FUNCTION_BLOCK FB_SystemControl
VAR_IN_OUT
	st_params								: ST_System_params;
	st_calibration							: ST_System_calibration;
	monitor								   	: ST_System_Monitor;
	control									: ST_System_Control;
END_VAR

VAR
	//fbs
	b_calibrationRunning					: BOOL;
	PowerControl							: FB_PowerControl;
	GenGridControl							: FB_GenGridController;
	r_trigStoreMachineSettings				: R_TRIG;
	
	b_skipPowerTest								: BOOL := TRUE;
	b_StoreMachineSettings						: BOOL;
	b_loadonly									: BOOL;
	sMessage									: STRING;	

	buffer										: ARRAY [0..24] OF WORD;		

END_VAR

VAR_OUTPUT
	toSystem								: ST_System_set();
END_VAR
VAR // added by the converter: edge detectors and wires of the graphical bodies
    _rt1, _rt2, _rt3 : R_TRIG;
    _w1, _w2 : BOOL;
END_VAR

//call methods
CalculateEfficiency(
	powerstack := monitor.powerstack, 
	powermonitor := monitor.powermonitor, 
	system := monitor.system,
	battery := monitor.battery);
	
FillSystemMonitoringVars();

MapUsercontrolsToSystemVars();

GetEvents();

//store machine settings
r_trigStoreMachineSettings(CLK := settings.Save OR settings.Load);
IF r_trigStoreMachineSettings.Q THEN
	b_StoreMachineSettings := TRUE;
END_IF

IF b_StoreMachineSettings AND_THEN storeSettings(TRUE, settings.Save) THEN;
	b_StoreMachineSettings := FALSE;
END_IF

//calibration script
IF NOT st_calibration.Powerstack.Slave.b_StartCalibration THEN
	PowerstackCalibration(start := st_calibration.Powerstack.Master.b_StartCalibration, skippowertest := b_skipPowerTest, loadonly := b_loadonly,   
		powerstack := monitor.powerstack,
		powermoduleCalib := st_calibration.Powerstack.Master,
		PMeasured := monitor.powermonitor.OutputField.ar_ActivePower[0],
		QMeasured := monitor.powermonitor.OutputField.ar_ReactivePower[0],
		sMessage => sMessage);
ELSIF NOT st_calibration.Powerstack.Master.b_StartCalibration THEN
	PowerstackCalibration(start := st_calibration.Powerstack.Slave.b_StartCalibration, skippowertest := b_skipPowerTest, loadonly := b_loadonly,   
		powerstack := monitor.powerstack,
		powermoduleCalib := st_calibration.Powerstack.Slave,
		PMeasured := monitor.powermonitor.OutputField.ar_ActivePower[0],
		QMeasured := monitor.powermonitor.OutputField.ar_ReactivePower[0],
		sMessage => sMessage);
END_IF
b_calibrationRunning := settings.Calibration.Powerstack.Master.b_StartCalibration OR settings.Calibration.Powerstack.Slave.b_StartCalibration;


UpdateSystemTime();

METHOD PRIVATE CalculateEfficiency : BOOL
VAR_IN_OUT
	powerstack 				: st_Powerstack_get;
	powermonitor			: st_powermonitor_get;
	system					: ST_system_get;
	battery					: ST_bms_get;
END_VAR

VAR_INST
	r_RawEfficiency	: REAL;
	r_AverageEfficiency: REAL;
	r_RoundtripEfficiency: REAL;
	
	
	ton_SumTimer			: TON :=(PT := T#100ms);
	r_EfficiencySum			: REAL;
	w_AverageSumCounter			: WORD;
END_VAR
r_RawEfficiency := ABS(powerstack.r_DCPower) / MAX(1,ABS(powermonitor.InputField.ar_ActivePower[0] + powermonitor.OutputField.ar_ActivePower[0])) * 100;

system.r_CurrentEfficiency := LIMIT(0, r_rawEfficiency, 99.8);

//manual averaging of the last hour of operation
ton_SumTimer(IN := NOT ton_SumTimer.Q);
IF powerstack.b_StartedState AND ton_SumTimer.Q THEN
	//reset counter and sum after 3000 samples +- 5min.
	IF w_AverageSumCounter = 3000 THEN
		//increment array index to add new efficiency value until upperbound has been reached.
		r_efficiencySum := r_efficiencySum - r_AverageEfficiency + system.r_CurrentEfficiency;
	ELSE
		//add new value to the summation
		w_AverageSumCounter := w_AverageSumCounter +1;
		r_EfficiencySum := r_efficiencySum + system.r_CurrentEfficiency;
	END_IF
	
	//System average efficiency during operation
	r_AverageEfficiency := r_EfficiencySum / MAX(1, w_AverageSumCounter);
	system.r_AvgEfficiency := r_AverageEfficiency;
	r_RoundtripEfficiency := LIMIT(0, powermonitor.Inverter.r_EnergySupplied / MAX(1,powermonitor.Inverter.r_EnergyConsumed - Battery.BatteryInfo.r_RemainingDischargeEnergyNett) * 100, 99);
	System.r_RoundtripEfficiency := r_RoundtripEfficiency;
END_IF
END_METHOD

METHOD ConfigureOutputContact : BOOL
VAR_INPUT
	SignalSelect			: eOutputContactSignal;
	GensetStartStop			: BOOL;
END_VAR
CASE SignalSelect OF
	eOutputContactSignal.FireAlarm 		: ConfigureOutputContact:= monitor.protections.FireDetection.b_FireAlarm;
	eOutputContactSignal.GenStartStop 	: ConfigureOutputContact:= GensetStartStop;
END_CASE
END_METHOD

METHOD EMstop : BOOL
VAR_INPUT
END_VAR

VAR_INST
	ton_FBdelay : TON := (PT:= T#20MS);
END_VAR
EMstop := FALSE;
ton_FBdelay(IN:= TRUE);

IF ton_FBdelay.Q THEN
	ton_FBdelay.IN := FALSE;
	EMstop := TRUE;
END_IF
END_METHOD

METHOD FillSystemMonitoringVars : BOOL

VAR_INST
	st_Params_MA			: ST_CTRL_MOVING_AVERAGE_PARAMS;
	ui_filterSize			: UINT := 50;
	fb_AverageEff			: FB_CTRL_MOVING_AVERAGE;
END_VAR
monitor.b_modeSwitchEnable := monitor.system.e_State = eSystemstate.Off OR 
	monitor.system.e_State = eSystemstate.StandBy OR
	monitor.system.e_State = eSystemstate.Init OR
	monitor.system.e_State = eSystemstate.Conditioning OR
	monitor.system.e_State = eSystemstate.Transport OR 
	monitor.system.e_State = eSystemstate.Dehumidifying OR
	monitor.system.e_State = eSystemState.EMstop; 

//Effiencies
monitor.system.b_StartAllowed := 
	control.HardSettings.system.e_EarthingSystem <> 0 AND
	monitor.powerstack.b_StartEnabled AND monitor.Cooling.ui_DehumRemainingTime = 0;
monitor.system.s_SystemName := Monitor.Router.Mobile.s_EmergencySMSDevName;

CASE toSystem.powerstack.e_Powermode OF
	ePowermodes.Droop: monitor.system.e_UgridPowermode := eUgridPowermode.Droop;
	ePowermodes.DroopZeroStart: monitor.system.e_UgridPowermode := eUgridPowermode.DroopZeroStart;
	ePowermodes.Isochronous: monitor.system.e_UgridPowermode := eUgridPowermode.Isochronous;
END_CASE

CASE toSystem.powerstack.e_InverterMode OF
	eInvertermodes.Afe : 
		monitor.system.e_gridmode := eGridmode.following;
		monitor.system.e_UgridPowermode := eUgridPowermode.None;
	eInvertermodes.Microgrid : monitor.system.e_gridmode := eGridmode.forming;
END_CASE
END_METHOD

METHOD GetDiagnostics
VAR_IN_OUT
	AddError		: ARRAY [*] OF FB_AddErrorST;
	a_ActiveEvents	: ARRAY [*] OF ST_ErrorStruct;
	w_Index			: WORD;
END_VAR
GenGridControl.GetDiagnostics(AddError, a_ActiveEvents, w_Index);
PowerControl.GetDiagnostics(AddError, a_ActiveEvents, w_Index);

(*Machine name update pending*) 	AddError[w_Index](
		b_ErrorTrig				:= monitor.system.events.b_RestartRequiredMachineName,
		out_ST_Error			:= a_ActiveEvents[w_Index],
		w_ErrorID				:= 1,
		e_ObjectID				:= eObject_ID.system,
		s_Message				:= 'Machinename update pending in VDL Powernet: System restart required',
		e_sev					:= eseverity.Info
		);
	w_Index := w_Index +1;
	
(*Machine name update pending*) AddError[w_Index](
		b_ErrorTrig				:= monitor.HartingIO.b_ExtSystemShutdownRequest,
		out_ST_Error			:= a_ActiveEvents[w_Index],
		w_ErrorID				:= 2,
		e_ObjectID				:= eObject_ID.system,
		s_Message				:= 'External IO initiated system shutdown',
		e_sev					:= eseverity.NormalShutdown,
		b_autoclear				:= FALSE
		);
	w_Index := w_Index +1;
	
(*time update failed*)	AddError[w_Index](
			b_ErrorTrig				:= monitor.system.events.b_TimeUpdateFailed,
			b_SMSEnableVDL			:= FALSE,
			out_ST_Error			:= a_ActiveEvents[w_Index],
			w_ErrorID				:= 3,					
			s_Message				:= 'System time update failed',
			e_sev					:= eSeverity.info,
			b_AutoClear				:= TRUE,
			e_ErrAckAccess			:= eErrAckAccess.General
			);
		w_Index := w_Index +1;
END_METHOD

METHOD GetEvents : BOOL
VAR_INPUT
END_VAR

VAR_INST
	s_machineNameOld : STRING;
	initdone		: BOOL;
END_VAR
IF NOT initdone AND monitor.system.s_SystemName <> '' THEN
	s_machineNameOld := monitor.system.s_SystemName;
	initdone := TRUE;
END_IF

monitor.system.events.b_RestartRequiredMachineName := s_machineNameOld <> monitor.system.s_SystemName;
END_METHOD

METHOD JsonFileToStruct : BOOL
VAR_INPUT
	bExecute			: BOOL;
	sJsonPathname		: STRING := 'C:\PLC_Utility\CalData_Powerstack.json';
	sStructName			: STRING;
	pStruct				: PVOID;
	nStruct				: UDINT;
	WriteMode			: BOOL;
	
END_VAR

VAR_OUTPUT
	Busy			: BOOL;
	Error			: BOOL;
	sMessage		: STRING;
END_VAR

VAR_INST
	bEnableCreateFile 	: BOOL := TRUE;
	SfcstepPrev		: BYTE;
	SFCTransAllowed	: BOOL;
	tofSFCstepDelay	: TOF := (PT := T#20MS);
	fbFileRead 		: FB_FileRead;
	fbFileWrite		: FB_FileWrite;
	fbFileOpen		: FB_FileOpen;
	fbFileClose		: FB_FileClose;
	sErrorMessage	: STRING;
	bLoading 		: BOOL;
	ton_executedelay	: TON := (PT := T#10MS);
	SFCstep			: BYTE;
	bLoad			: BOOL;
	bError			: BOOL;
	bfileOpened		: BOOL;
	hrErrorCode		: HRESULT;
	fbJson         : FB_JsonSaxWriter;
  	fbJsonDataType : FB_JsonReadWriteDataType;
  	sJsonDoc     	: STRING(10000);
	nBytesRead		: UDINT;
	b_CreateNewFile 	: BOOL;
	bOpenExecute		: BOOL;
	bReadExecute		: BOOL;
	bWriteExecute		: BOOL;
	bCloseExecute		: BOOL;
	nModeSel			: DWORD;	
	udLength			: UDINT;
	tDelayWriting		: TON := (PT := T#50MS);
	bEnable : BOOL := FALSE;
	
END_VAR
 

IF NOT ton_executedelay.Q THEN
	sfcstep := 0;
END_IF

IF pStruct = 0 THEN
	sfcstep := 99;
	sErrorMessage := 'Invalid pointer to struct';
ELSIF nStruct = 0 THEN
	sfcstep := 99;
	sErrorMessage := 'Invalid size of struct';
END_IF

//transition delay logic.
tofSFCstepDelay(IN := SFCstep <> SFCstepPrev);
SFCTransAllowed := NOT tofSFCstepDelay.Q AND bLoading;

CASE SFCstep OF
0: //idle
bEnable := FALSE;
	bLoading := FALSE;
	bError := FALSE;
	SFCTransAllowed := FALSE;
	bOpenExecute 			:= FALSE;
	bReadExecute 			:= FALSE;
	bWriteExecute 			:= FALSE;
	bCloseExecute 			:= FALSE;
	bEnableCreateFile 		:= FALSE;
	
	ton_executedelay(IN := bExecute);
	
	IF ton_executedelay.Q THEN
		sfcstep := SEL(writemode OR b_CreateNewFile, 1, 2);
		nModeSel 		:= SEL(sfcstep = 1, FOPEN_MODEWRITE,FOPEN_MODEREAD);
		sErrorMessage := '';
		bLoading := TRUE;	
	END_IF
	
1: 	//open file
	sJsonDoc := '';
	nModeSel 				:= FOPEN_MODEREAD;
	bReadExecute 			:= FALSE;
	bWriteExecute 			:= FALSE;
	bCloseExecute 			:= FALSE;
	bOpenExecute 			:= SFCTransAllowed;
	
	
	IF bEnable THEN 
	//IF SFCTransAllowed THEN
		IF fbFileOpen.hfile <> 0 AND NOT fbFileOpen.bBusy AND NOT fbFileOpen.bError THEN
			SFCstep := 10;
			bEnable := FALSE;
		ELSIF fbFileOpen.bError THEN
			sErrorMessage := CONCAT('Error opening file: sfc step ', TO_STRING(sfcstep));
			sfcstep := SEL(bEnableCreateFile, 97, 2);
		END_IF
	END_IF
	
2: //create file if non existing
	sJsonDoc := '';
	b_createNewFile := FALSE;
	nModeSel 				:= FOPEN_MODEWRITE;
	bReadExecute 			:= FALSE;
	bWriteExecute 			:= FALSE;
	bCloseExecute 			:= FALSE;
	bOpenExecute 			:= SFCTransAllowed;

	
	IF bEnable THEN 
		IF fbFileOpen.hfile <> 0 AND NOT fbFileOpen.bBusy AND NOT fbFileOpen.bError THEN
			sErrorMessage := 'New file created';
			sJsonDoc 		:= '';
			MEMSET(ADR(sJsonDoc), 0, SIZEOF(sJsonDoc));
			SFCstep := 3;
			bEnable := FALSE;
		ELSIF fbFileOpen.bError THEN
			sErrorMessage := CONCAT('Error opening and creating file: sfc step ', TO_STRING(sfcstep));
			sfcstep := 97;
		END_IF
	END_IF
	
3: //Write current struct values to new Json string
//	IF LEN(sJsonDoc) = 0 THEN
		fbJson.ResetDocument();
		fbJsonDataType.AddJsonValueFromSymbol(fbJson, sStructName, nStruct, pStruct, hrErrorCode => hrErrorCode);
		udLength := fbJson.GetDocumentLength();
		fbJson.CopyDocument(sJsonDoc, udLength);
//	END_IF
	
	IF SFCTransAllowed THEN
		IF hrErrorCode = 0 THEN
			bError := FALSE;
			sfcstep := 4; //final step
		ELSE
			bError := TRUE;
			sErrorMessage := CONCAT('Error generating json string: SFC step ', TO_STRING(sfcstep));
			sfcstep := 97; //error step
		END_IF
	END_IF
	
4: //write json string to file
	bReadExecute 	:= FALSE;
	bOpenExecute 	:= FALSE;
	bCloseExecute 	:= FALSE;
	bWriteExecute 	:= SFCTransAllowed;
	
	IF SFCTransAllowed THEN
		IF NOT fbFileWrite.bBusy AND NOT fbFileWrite.bError THEN
			SFCstep := 97;
			bEnable := FALSE;
		ELSIF fbFileWrite.bError THEN
			sErrorMessage := CONCAT('Error writing file: sfc step ', TO_STRING(sfcstep));
			sfcstep := 97;
		END_IF
	END_IF
		
10: //Read File
	sJsonDoc 		:= '';
	bOpenExecute 	:= FALSE;
	bWriteExecute 	:= FALSE;
	bCloseExecute 	:= FALSE;
	bReadExecute 	:= SFCTransAllowed;
	
	IF SFCTransAllowed THEN
		IF NOT fbFileRead.bBusy AND NOT fbFileRead.bError THEN
			SFCstep := 11;
			bEnable := FALSE;
		ELSIF fbFileRead.bError THEN
			sErrorMessage := CONCAT('Error reading file: sfc step ', TO_STRING(sfcstep));
			sfcstep :=  97;
			b_createNewFile := bEnableCreateFile;
		END_IF
	END_IF

	
11: //Convert buffer to struct
	fbJsonDataType.SetSymbolFromJson(sJsonDoc, sStructName, nStruct, pStruct, hrErrorCode => hrErrorCode);
	
	IF SFCTransAllowed THEN
		
		IF hrErrorCode = 0 THEN
			bError := FALSE;
			sfcstep := 97; //final step
		ELSE
			bError := TRUE;
			sErrorMessage := CONCAT('Error writing file to struct: sfc step ', TO_STRING(sfcstep));
			sfcstep := 97;
			b_createNewFile := bEnableCreateFile;	
		END_IF
	END_IF

97: // file opened
	
	bWriteExecute 	:= FALSE;
	bOpenExecute 	:= FALSE;
	bReadExecute 	:= FALSE;
	bCloseExecute 	:= bfileOpened := fbFileOpen.hFile <> 0;

	
	IF SFCTransAllowed THEN
		IF NOT fbFileClose.bBusy AND NOT fbFileClose.bError THEN
			bfileOpened := FALSE;
			sfcstep := 98;
			bEnable := FALSE;
		ELSIF fbFileClose.bError THEN
			sErrorMessage := CONCAT('Error closing file ', TO_STRING(sfcstep));
			bError := TRUE;
			sfcstep := 98;
		END_IF
	END_IF
	
98: 	//feedback and reset method for next request
	IF NOT bError THEN
		sErrorMessage := 'SUCCES';
	ELSE
		Error := TRUE;
	END_IF
	bEnable := FALSE;
	bOpenExecute 		:= FALSE;
	bReadExecute 		:= FALSE;
	bWriteExecute 		:= FALSE;
	bCloseExecute 		:= FALSE;
	ton_executedelay.IN := FALSE;
	sfcstep := 99;
	
	
99: //once here, reset SFC
	IF NOT b_CreateNewFile THEN
		JsonFileToStruct := TRUE;
	END_IF
	sfcstep := 0;
END_CASE
	


fbFileOpen(sPathName:= sJsonPathname , nMode := nModeSel ,bExecute:= bOpenExecute);
fbFileWrite(hFile := fbFileOpen.hFile , pWriteBuff := ADR(sJsonDoc),bExecute := bWriteExecute , cbWriteLen := udLength);
fbFileRead(hFile := fbFileOpen.hFile, pReadBuff := ADR(sJsonDoc), cbReadLen := SIZEOF(sJsonDoc),bExecute := bReadExecute, cbRead => nBytesRead);
fbFileClose(hFile := fbFileOpen.hFile, bExecute := bCloseExecute);

IF fbFileOpen.bBusy AND bOpenExecute THEN
	bOpenExecute := FALSE;
	bEnable := TRUE;
END_IF
//	rTrigExecute(CLK := FALSE);
//	IF NOT rTrigExecute.CLK THEN
//		JsonFileToStruct := TRUE;
SFCstepPrev := SFCstep;

//output data
busy := bLoading;
sMessage := sErrorMessage;
END_METHOD

ACTION Map_ACDCchargerControls:
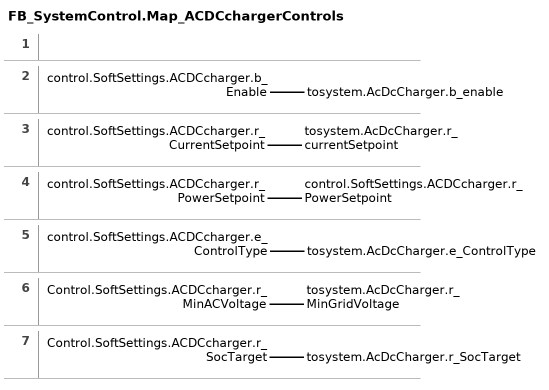
// NETWORK 1

// NETWORK 2
tosystem.AcDcCharger.b_enable := control.SoftSettings.ACDCcharger.b_Enable;

// NETWORK 3
tosystem.AcDcCharger.r_currentSetpoint := control.SoftSettings.ACDCcharger.r_CurrentSetpoint;

// NETWORK 4
control.SoftSettings.ACDCcharger.r_PowerSetpoint := control.SoftSettings.ACDCcharger.r_PowerSetpoint;

// NETWORK 5
tosystem.AcDcCharger.e_ControlType := control.SoftSettings.ACDCcharger.e_ControlType;

// NETWORK 6
tosystem.AcDcCharger.r_MinGridVoltage := Control.SoftSettings.ACDCcharger.r_MinACVoltage;

// NETWORK 7
tosystem.AcDcCharger.r_SocTarget := Control.SoftSettings.ACDCcharger.r_SocTarget;
END_ACTION

ACTION MaP_BMSControl:
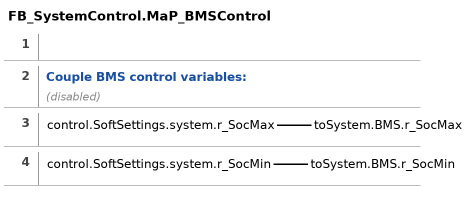
// NETWORK 1

// NETWORK 2 (disabled)
// label: Couple BMS control variables

// NETWORK 3
toSystem.BMS.r_SocMax := control.SoftSettings.system.r_SocMax;

// NETWORK 4
toSystem.BMS.r_SocMin := control.SoftSettings.system.r_SocMin;
END_ACTION

ACTION Map_DCLink:
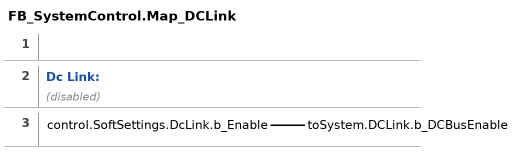
// NETWORK 1

// NETWORK 2 (disabled)
// label: Dc Link

// NETWORK 3
toSystem.DCLink.b_DCBusEnable := control.SoftSettings.DcLink.b_Enable;
END_ACTION

ACTION Map_GenCommControls:
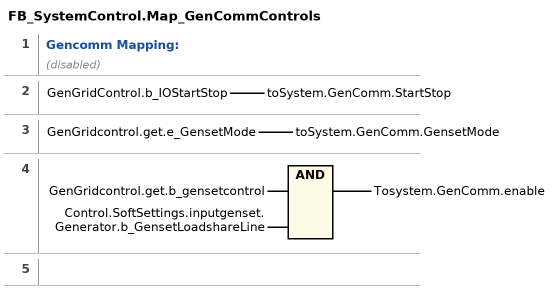
// NETWORK 1 (disabled)
// label: Gencomm Mapping

// NETWORK 2
toSystem.GenComm.StartStop := GenGridControl.b_IOStartStop;

// NETWORK 3
toSystem.GenComm.GensetMode := GenGridcontrol.get.e_GensetMode;

// NETWORK 4
Tosystem.GenComm.enable := GenGridcontrol.get.b_gensetcontrol AND Control.SoftSettings.inputgenset.Generator.b_GensetLoadshareLine;

// NETWORK 5
END_ACTION

ACTION Map_GeneralControls:
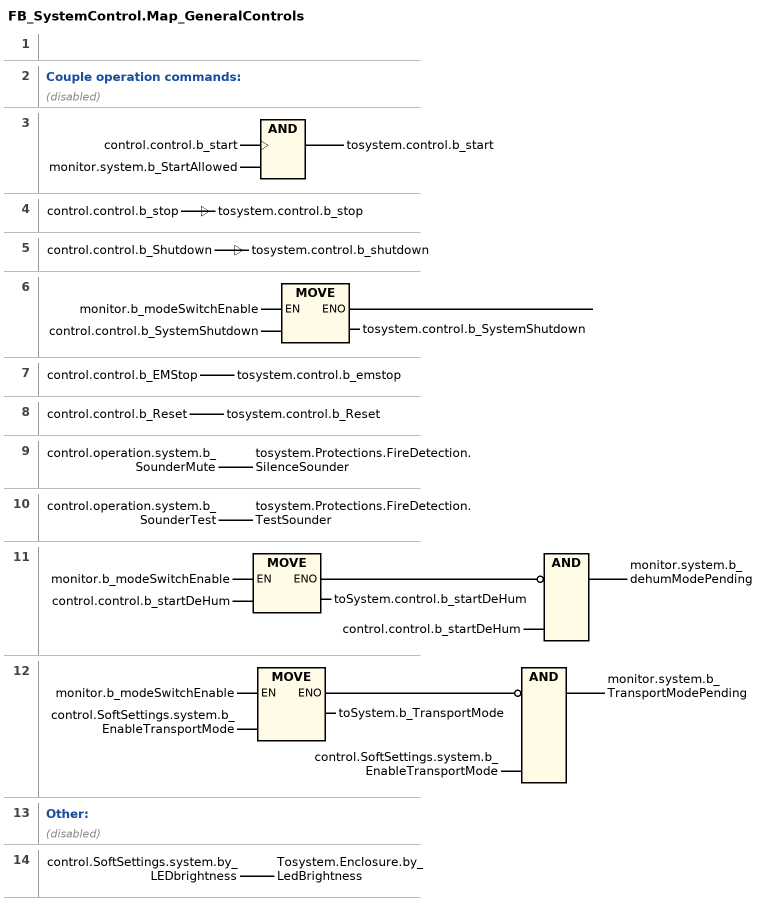
// NETWORK 1

// NETWORK 2 (disabled)
// label: Couple operation commands

// NETWORK 3
_rt1(CLK := control.control.b_start);
tosystem.control.b_start := _rt1.Q AND monitor.system.b_StartAllowed;

// NETWORK 4
_rt2(CLK := control.control.b_stop);
tosystem.control.b_stop := _rt2.Q;

// NETWORK 5
_rt3(CLK := control.control.b_Shutdown);
tosystem.control.b_shutdown := _rt3.Q;

// NETWORK 6
IF monitor.b_modeSwitchEnable THEN tosystem.control.b_SystemShutdown := control.control.b_SystemShutdown; END_IF

// NETWORK 7
tosystem.control.b_emstop := control.control.b_EMStop;

// NETWORK 8
tosystem.control.b_Reset := control.control.b_Reset;

// NETWORK 9
tosystem.Protections.FireDetection.SilenceSounder := control.operation.system.b_SounderMute;

// NETWORK 10
tosystem.Protections.FireDetection.TestSounder := control.operation.system.b_SounderTest;

// NETWORK 11
_w1 := monitor.b_modeSwitchEnable;
IF _w1 THEN toSystem.control.b_startDeHum := control.control.b_startDeHum; END_IF
monitor.system.b_dehumModePending := NOT _w1 AND control.control.b_startDeHum;

// NETWORK 12
_w2 := monitor.b_modeSwitchEnable;
IF _w2 THEN toSystem.b_TransportMode := control.SoftSettings.system.b_EnableTransportMode; END_IF
monitor.system.b_TransportModePending := NOT _w2 AND control.SoftSettings.system.b_EnableTransportMode;

// NETWORK 13 (disabled)
// label: Other

// NETWORK 14
Tosystem.Enclosure.by_LedBrightness := control.SoftSettings.system.by_LEDbrightness;
END_ACTION

ACTION Map_HartingIO:
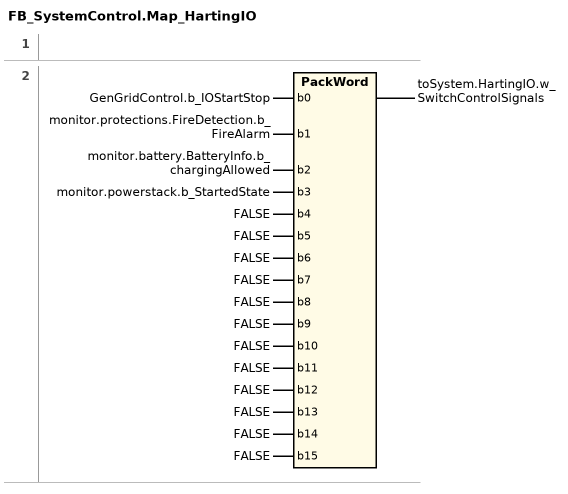
// NETWORK 1

// NETWORK 2
toSystem.HartingIO.w_SwitchControlSignals := PackWord(b0 := GenGridControl.b_IOStartStop, b1 := monitor.protections.FireDetection.b_FireAlarm, b2 := monitor.battery.BatteryInfo.b_chargingAllowed, b3 := monitor.powerstack.b_StartedState, b4 := FALSE, b5 := FALSE, b6 := FALSE, b7 := FALSE, b8 := FALSE, b9 := FALSE, b10 := FALSE, b11 := FALSE, b12 := FALSE, b13 := FALSE, b14 := FALSE, b15 := FALSE);
END_ACTION

ACTION Map_PowerstackControls:
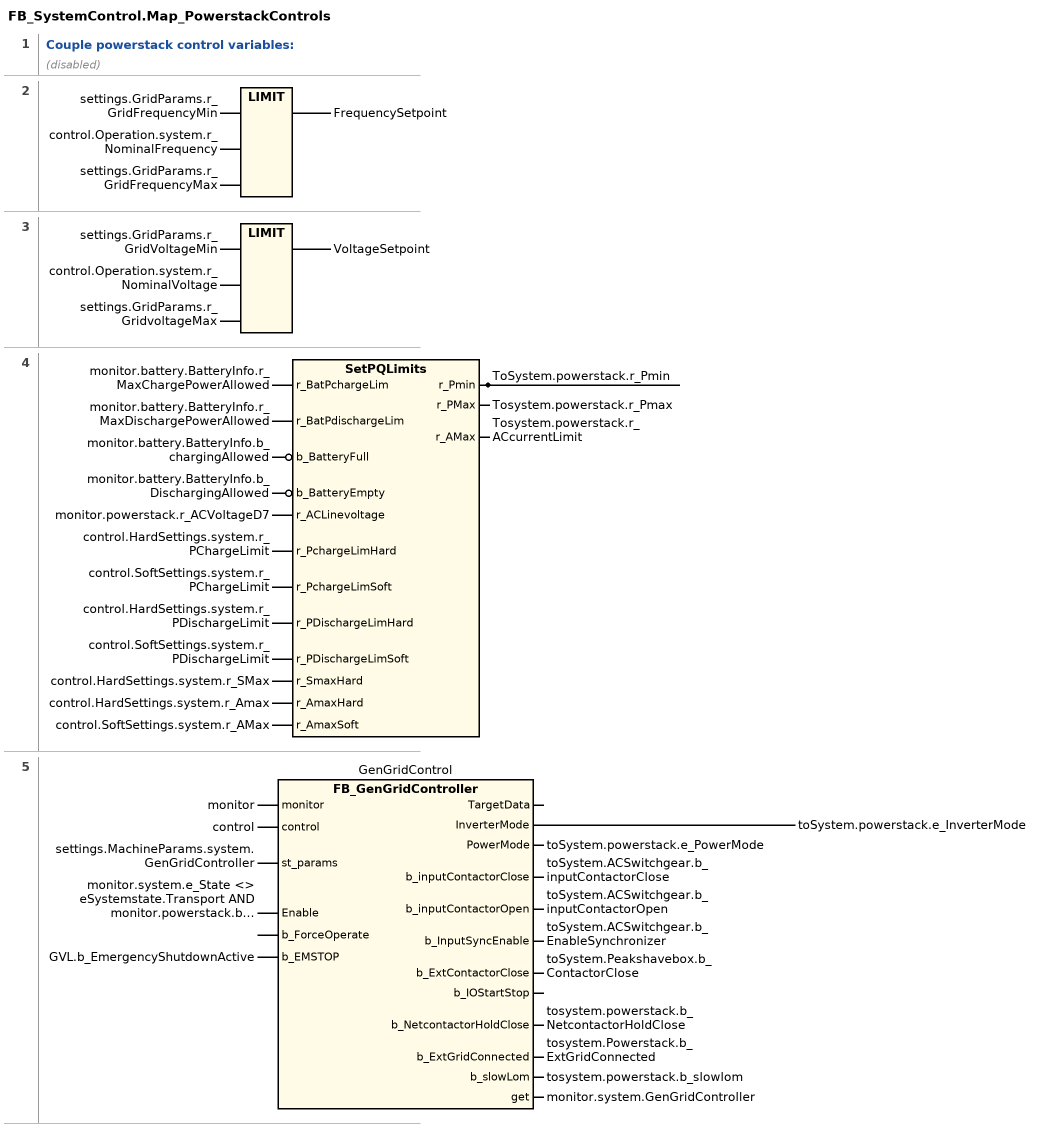
// NETWORK 1 (disabled)
// label: Couple powerstack control variables

// NETWORK 2
FrequencySetpoint := LIMIT(settings.GridParams.r_GridFrequencyMin, control.Operation.system.r_NominalFrequency, settings.GridParams.r_GridFrequencyMax);

// NETWORK 3
VoltageSetpoint := LIMIT(settings.GridParams.r_GridVoltageMin, control.Operation.system.r_NominalVoltage, settings.GridParams.r_GridvoltageMax);

// NETWORK 4
SetPQLimits(r_BatPchargeLim := monitor.battery.BatteryInfo.r_MaxChargePowerAllowed, r_BatPdischargeLim := monitor.battery.BatteryInfo.r_MaxDischargePowerAllowed, b_BatteryFull := NOT monitor.battery.BatteryInfo.b_chargingAllowed, b_BatteryEmpty := NOT monitor.battery.BatteryInfo.b_DischargingAllowed, r_ACLinevoltage := monitor.powerstack.r_ACVoltageD7, r_PchargeLimHard := control.HardSettings.system.r_PChargeLimit, r_PchargeLimSoft := control.SoftSettings.system.r_PChargeLimit, r_PDischargeLimHard := control.HardSettings.system.r_PDischargeLimit, r_PDischargeLimSoft := control.SoftSettings.system.r_PDischargeLimit, r_SmaxHard := control.HardSettings.system.r_SMax, r_AmaxHard := control.HardSettings.system.r_Amax, r_AmaxSoft := control.SoftSettings.system.r_AMax, r_Pmin => ToSystem.powerstack.r_Pmin, r_PMax => Tosystem.powerstack.r_Pmax, r_AMax => Tosystem.powerstack.r_ACcurrentLimit);

// NETWORK 5
GenGridControl(
    monitor := monitor,
    control := control,
    st_params := settings.MachineParams.system.GenGridController,
    Enable := monitor.system.e_State <> eSystemstate.Transport AND monitor.powerstack.b_ControlEnabled,
    b_EMSTOP := GVL.b_EmergencyShutdownActive,
    PowerMode => toSystem.powerstack.e_PowerMode,
    b_inputContactorClose => toSystem.ACSwitchgear.b_inputContactorClose,
    b_inputContactorOpen => toSystem.ACSwitchgear.b_inputContactorOpen,
    b_InputSyncEnable => toSystem.ACSwitchgear.b_EnableSynchronizer,
    b_ExtContactorClose => toSystem.Peakshavebox.b_ContactorClose,
    b_NetcontactorHoldClose => tosystem.powerstack.b_NetcontactorHoldClose,
    b_ExtGridConnected => tosystem.Powerstack.b_ExtGridConnected,
    b_slowLom => tosystem.powerstack.b_slowlom,
    get => monitor.system.GenGridController); // FB_GenGridController
toSystem.powerstack.e_InverterMode := GenGridControl.InverterMode;

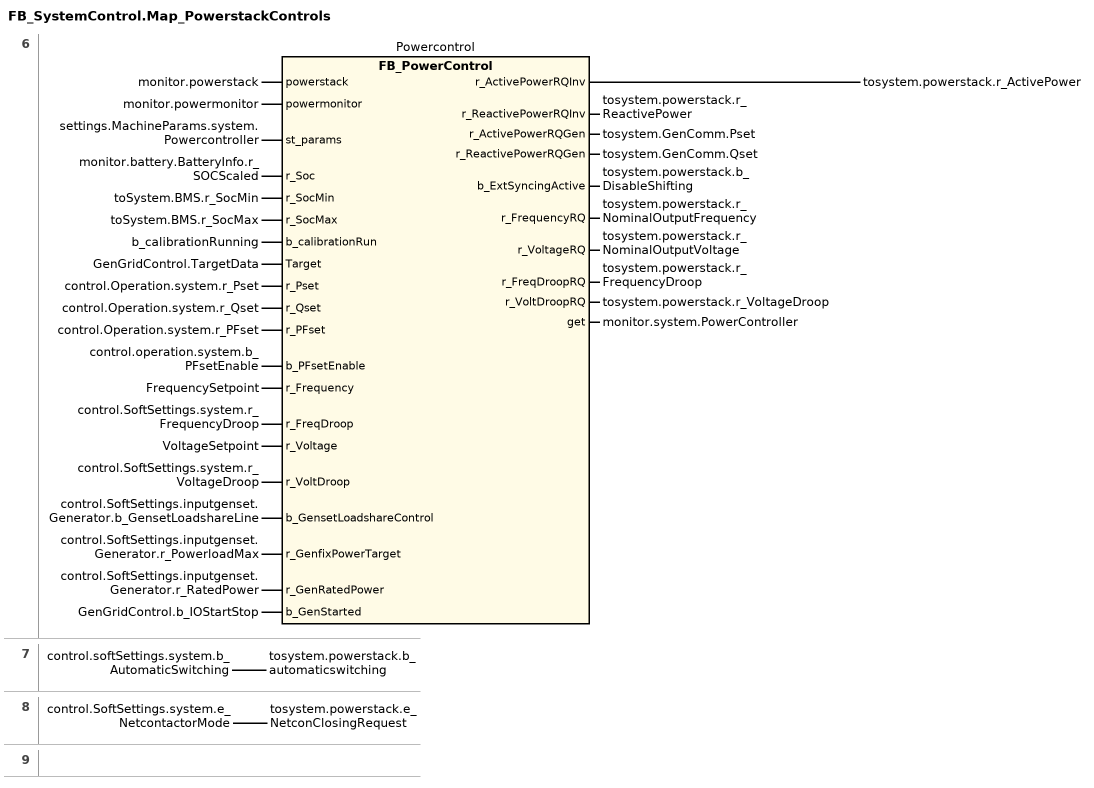
// NETWORK 6
Powercontrol(
    powerstack := monitor.powerstack,
    powermonitor := monitor.powermonitor,
    st_params := settings.MachineParams.system.Powercontroller,
    r_Soc := monitor.battery.BatteryInfo.r_SOCScaled,
    r_SocMin := toSystem.BMS.r_SocMin,
    r_SocMax := toSystem.BMS.r_SocMax,
    b_calibrationRun := b_calibrationRunning,
    Target := GenGridControl.TargetData,
    r_Pset := control.Operation.system.r_Pset,
    r_Qset := control.Operation.system.r_Qset,
    r_PFset := control.Operation.system.r_PFset,
    b_PFsetEnable := control.operation.system.b_PFsetEnable,
    r_Frequency := FrequencySetpoint,
    r_FreqDroop := control.SoftSettings.system.r_FrequencyDroop,
    r_Voltage := VoltageSetpoint,
    r_VoltDroop := control.SoftSettings.system.r_VoltageDroop,
    b_GensetLoadshareControl := control.SoftSettings.inputgenset.Generator.b_GensetLoadshareLine,
    r_GenfixPowerTarget := control.SoftSettings.inputgenset.Generator.r_PowerloadMax,
    r_GenRatedPower := control.SoftSettings.inputgenset.Generator.r_RatedPower,
    b_GenStarted := GenGridControl.b_IOStartStop,
    r_ReactivePowerRQInv => tosystem.powerstack.r_ReactivePower,
    r_ActivePowerRQGen => tosystem.GenComm.Pset,
    r_ReactivePowerRQGen => tosystem.GenComm.Qset,
    b_ExtSyncingActive => tosystem.powerstack.b_DisableShifting,
    r_FrequencyRQ => tosystem.powerstack.r_NominalOutputFrequency,
    r_VoltageRQ => tosystem.powerstack.r_NominalOutputVoltage,
    r_FreqDroopRQ => tosystem.powerstack.r_FrequencyDroop,
    r_VoltDroopRQ => tosystem.powerstack.r_VoltageDroop,
    get => monitor.system.PowerController); // FB_PowerControl
tosystem.powerstack.r_ActivePower := Powercontrol.r_ActivePowerRQInv;

// NETWORK 7
tosystem.powerstack.b_automaticswitching := control.softSettings.system.b_AutomaticSwitching;

// NETWORK 8
tosystem.powerstack.e_NetconClosingRequest := control.SoftSettings.system.e_NetcontactorMode;

// NETWORK 9
END_ACTION

ACTION Map_ProtectionSystemControls:
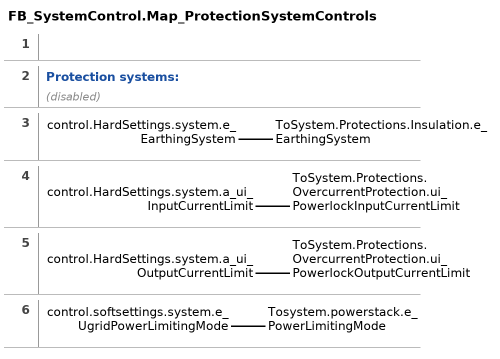
// NETWORK 1

// NETWORK 2 (disabled)
// label: Protection systems

// NETWORK 3
ToSystem.Protections.Insulation.e_EarthingSystem := control.HardSettings.system.e_EarthingSystem;

// NETWORK 4
ToSystem.Protections.OvercurrentProtection.ui_PowerlockInputCurrentLimit := control.HardSettings.system.a_ui_InputCurrentLimit;

// NETWORK 5
ToSystem.Protections.OvercurrentProtection.ui_PowerlockOutputCurrentLimit := control.HardSettings.system.a_ui_OutputCurrentLimit;

// NETWORK 6
Tosystem.powerstack.e_PowerLimitingMode := control.softsettings.system.e_UgridPowerLimitingMode;
END_ACTION

ACTION Map_PSBControls:
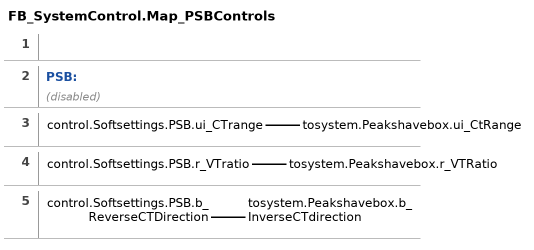
// NETWORK 1

// NETWORK 2 (disabled)
// label: PSB

// NETWORK 3
tosystem.Peakshavebox.ui_CtRange := control.Softsettings.PSB.ui_CTrange;

// NETWORK 4
tosystem.Peakshavebox.r_VTRatio := control.Softsettings.PSB.r_VTratio;

// NETWORK 5
tosystem.Peakshavebox.b_InverseCTdirection := control.Softsettings.PSB.b_ReverseCTDirection;
END_ACTION

METHOD MapUsercontrolsToSystemVars : BOOL
VAR_INPUT
END_VAR
Map_GeneralControls();
Map_PowerstackControls();
Map_ProtectionSystemControls();
Map_PSBControls();
Map_GenCommControls();
Map_BMSControl();
Map_ACDCChargerControls();
Map_HartingIO();
Map_DCLink();
END_METHOD

METHOD PowerstackCalibration : BOOL

VAR_INPUT
	start 						: BOOL;
	skippowertest				: BOOL;
	loadonly					: BOOL;
END_VAR

VAR_IN_OUT CONSTANT
	powerstack					: ST_Powerstack_get;
END_VAR


VAR_IN_OUT
	powermoduleCalib				: ST_Powermodule_Calibration;
END_VAR

VAR_IN_OUT CONSTANT
	PMeasured					: REAL;
	QMeasured					: REAL;
END_VAR

VAR_OUTPUT
	Error : BOOL;
	Busy : BOOL;
	sMessage : STRING;
END_VAR

VAR_INST
	PSetPoints : ARRAY[0..4] OF REAL := [-250, -125, 0, 125, 250];
    QSetPoints : ARRAY[0..4] OF REAL := [-250, -125, 0, 125, 250];
	
	fTrigStop					: f_TRIG;
	rTrigExecute				: r_trig;
	fbExecuteCalibrationFit 	: NT_StartProcess;
	bFileDeleted				: BOOL;
	fbFileDelete				: FB_FileDelete;
	ton_FileNotExising			: TON := (PT := T#60S);
	bError						: BOOL;
	bBusy						: BOOL;
	
	
	pulseTimer					: TON := (PT := T#1S);
	DelayTimer					: TON := (PT := T#5S);
	i 							: INT 			:=0;
	j 							: INT 			:=0;
	SFCstep						: INT;
	Message					: STRING;
END_VAR
// Pset+
IF NOT start THEN
	i 		:= 0;
	j 		:= 0;
END_IF

fTrigStop(CLK := start);
IF fTrigStop.Q THEN
	sfcstep := 99;
END_IF
	

CASE SFCstep OF
	0: 
		ton_FileNotExising(IN := FALSE);
		pulseTimer.IN := FALSE;
		DelayTimer(IN := FALSE);
		rTrigExecute(CLK := START);
		IF rTrigExecute.Q THEN
			IF loadonly THEN
				SFCstep := 4;
			ELSIF skippowertest THEN
				SFCstep := 2;
			ELSE
				SFCstep := 1; 
			END_IF
		END_IF
		
	1: // do calibration and get data
		powermoduleCalib.b_StartCalibration := start AND NOT powerstack.b_InverterGridFormingMode AND powerstack.b_StartedState;
		DelayTimer(IN:=NOT delaytimer.Q AND start);
		powermoduleCalib.CalibrationData.Pset[i]:= powermoduleCalib.r_Pset;
		powermoduleCalib.CalibrationData.Qset[j] := powermoduleCalib.r_Qset;
		powermoduleCalib.r_Pset := PSetPoints[i];
		powermoduleCalib.r_Qset := QSetPoints[j];
		IF delaytimer.Q THEN
			j := j +1;
			
			IF j = 5 THEN
				i := i +1;
				j := 0;
				IF i = 5 THEN
					i 		:= 0;
					j 		:= 0;
					powermoduleCalib.r_Pset := 0;
					powermoduleCalib.r_Qset := 0;
					sfcstep := 2;
					RETURN;
				END_IF
			END_IF
		END_IF
		powermoduleCalib.CalibrationData.Pmeas[i][j] := PMeasured;
		powermoduleCalib.CalibrationData.Qmeas[i][j] := QMeasured;

	
	2:	//export data to json
		powermoduleCalib.b_StartCalibration := TRUE;
		pulseTimer(IN := NOT JsonFileToStruct(
			bExecute := pulseTimer.Q,
			sJsonPathName := 'C:\PLCUtility\CalDat_Powerstack.json',
			sStructName := 'ST_Powerstack_Calibration',
			pStruct := ADR(st_calibration.Powerstack),
			nStruct := SIZEOF(st_calibration.Powerstack),
			WriteMode := TRUE,
			sMessage => Message
			));
		IF NOT pulseTimer.IN THEN
			SFCstep := 3;
		END_IF
	3: //execute calibration python script
		fbExecuteCalibrationFit(
			NETID		:= '',
			PATHSTR		:= 'C:\PLCUtility\CalibrationFit.exe',
			DIRNAME		:= 'C:\PLCUtility',
			START		:= TRUE,
			COMNDLINE	:= '',
			TMOUT		:= T#60S,
			BUSY		=> bBusy,
			ERR			=> bError
		);
		
		ton_FileNotExising(IN := TRUE);
		pulseTimer(IN := NOT fbFileDelete.bExecute AND NOT fbFileDelete.bBusy);
		fbFileDelete(
			sPathName := 'C:\PLCUtility\caliblog.txt');
		fbFileDelete.bExecute := pulsetimer.Q;

		IF fbFileDelete.bExecute AND NOT fbFileDelete.bBusy THEN
			bFileDeleted := NOT fbFileDelete.bERROR;
		END_IF
		
		IF bFileDeleted THEN
			bFileDeleted := FALSE;	
			SFCstep := 4;
			pulseTimer.IN := FALSE;
		ELSIF bError OR ton_FileNotExising.Q THEN
			SFCstep := 99;
		END_IF
	
	4: //Read back calibration file
		powermoduleCalib.b_StartCalibration := FALSE;
		pulseTimer(IN := NOT JsonFileToStruct(
			bExecute := pulseTimer.Q,
			sJsonPathName := 'C:\PLCUtility\CalDat_Powerstack.json',
			sStructName := 'ST_Powerstack_Calibration',
			pStruct := ADR(st_calibration.Powerstack),
			nStruct := SIZEOF(st_calibration.Powerstack),
			WriteMode := FALSE,
			sMessage => Message,
			Error => bError,
			Busy => bBusy
			));
		IF NOT pulseTimer.IN THEN
			SFCstep := 99;
		END_IF
		
	99: //clear all states for next round
		Error := bError; 
		sMessage := Message;
		pulseTimer.IN := FALSE;
		fbExecuteCalibrationFit(START := FALSE);
		DelayTimer.IN := FALSE;
		fbExecuteCalibrationFit.START := FALSE;
		PowerstackCalibration := TRUE;
		SFCstep := 0;
END_CASE
END_METHOD

METHOD Reset : BOOL
Reset := GenGridControl.Reset();
END_METHOD

METHOD SetPQLimits

VAR_INPUT
	r_BatPchargeLim			: REAL;
	r_BatPdischargeLim		: REAL;
	b_BatteryFull			: BOOL;
	b_BatteryEmpty			: BOOL;
	r_ACLinevoltage			: REAL;
	r_PchargeLimHard		: REAL;
	r_PchargeLimSoft		: REAL;
	r_PDischargeLimHard		: REAL;
	r_PDischargeLimSoft		: REAL;
	r_SmaxHard				: REAL;	//kVA
	r_AmaxHard				: REAL; //current
	r_AmaxSoft				: REAL; //current
END_VAR

VAR_OUTPUT
	r_Pmin				: REAL;
	r_PMax				: REAL;
	r_AMax				: REAL;
END_VAR

VAR_INST
	fb_rampPcharge						: FB_ramp := (b_enable := TRUE, r_ramprate := 25);
	fb_rampPdischarge					: FB_ramp := (b_enable := TRUE, r_ramprate := 25);
	fb_rampCurrentLimit					: FB_ramp := (b_enable := TRUE, r_ramprate := 100);
	
	r_BatChargeCorrectionFactor			: REAL := 0.98; // compensates inverter losses and BMS measurement errors
	r_BatDischargeCorrectionFactor		: REAL := 0.99;
	r_Smax								: REAL;
	r_PDischargeLimitUser				: REAL; //Discharging
	r_PChargeLimitUser					: REAL; //Charging
	r_AmaxLimitUser						: REAL;
	r_PmaxbySmax						: REAL;
	r_BatChargePowerLimitCalc			: REAL;
	r_BatDischargePowerLimitCalc		: REAL;
END_VAR
//user soft limit
fb_rampPcharge(IN := LIMIT(0 ,r_PchargeLimSoft, r_PchargeLimHard));
fb_rampPdischarge(IN := LIMIT(0,r_PDischargeLimSoft, r_PDischargeLimHard));

//current limit
r_AmaxLimitUser := MAX(0, KwToCurrent(r_SmaxHard,r_acLineVoltage), r_AmaxHard);
fb_rampCurrentLimit(IN := LIMIT(0,r_Amaxsoft, r_AmaxLimitUser), Q=> r_AMax);

r_Smax:= CurrentToKw(r_Amax, r_AClinevoltage);
r_PmaxbySmax := r_SMax; //SQRT(MAX(EXPT(r_Smax,2) - EXPT(r_ReaPower, 2),0));

//Set system Variable
r_Pmin := -MIN(ABS(r_BatPchargeLim / r_BatChargeCorrectionFactor), fb_rampPcharge.Q, r_PmaxbySmax);
r_Pmax := MIN(ABS(r_BatPdischargeLim * r_BatDischargeCorrectionFactor),  fb_rampPdischarge.Q, r_PmaxbySmax);

IF b_BatteryFull THEN
	r_Pmin := 0;
ELSIF b_BatteryEmpty THEN
	r_Pmax := 0; //overwrite value from input to 0.
END_IF
END_METHOD

METHOD shutdown : BOOL
VAR_INPUT
END_VAR

VAR_INST
	started : BOOL;
	ton_RetryDelay : TON := (PT := T#2s);
END_VAR
ton_RetryDelay(IN := TRUE);

IF storeSettings(ton_RetryDelay.Q, FALSE) THEN
	shutdown := TRUE;
	ton_RetryDelay(IN := FALSE);
END_IF
END_METHOD

METHOD StoreSettings : BOOL
VAR_INPUT
	execute : BOOL;
	writeMode: BOOL;
END_VAR

VAR_INST
	rTrigExecute	: R_TRIG;
	b_next : BOOL;
	sfcStep	: BYTE;
	tDelaySFCstep		: TON :=(PT := T#10MS);
END_VAR
rTrigExecute(CLK := execute);
IF rTrigExecute.Q THEN
	SFCstep := 1;
END_IF

CASE SFCstep OF
	1: b_next := JsonFileToStruct(
		bExecute := TRUE,
		sJsonPathName := 'C:\PLCUtility\MachineSettings.json',
		sStructName := 'ST_System_MachineParams',
		pStruct := ADR(settings.MachineParams),
		nStruct := SIZEOF(settings.MachineParams),
		WriteMode := writeMode,
		sMessage => sMessage
		);
	2: b_next := JsonFileToStruct(
		bExecute := TRUE,
		sJsonPathName := 'C:\PLCUtility\MachineConfig.json',
		sStructName := 'ST_System_Config',
		pStruct := ADR(settings.Configuration),
		nStruct := SIZEOF(settings.Configuration),
		WriteMode := writeMode,
		sMessage => sMessage
		);
	 3: b_next := JsonFileToStruct(
		bExecute := TRUE,
		sJsonPathName := 'C:\PLCUtility\GridSettings.json',
		sStructName := 'ST_System_GridCodeParams',
		pStruct := ADR(settings.GridParams),
		nStruct := SIZEOF(settings.GridParams),
		WriteMode := writeMode,
		sMessage => sMessage
		);
	 4: b_next := JsonFileToStruct(
		bExecute := TRUE,
		sJsonPathName := 'C:\PLCUtility\MachineProperties.json',
		sStructName := 'ST_System_Properties',
		pStruct := ADR(settings.Properties),
		nStruct := SIZEOF(settings.Properties),
		WriteMode := writeMode,
		sMessage => sMessage
		);
	5: b_next := JsonFileToStruct(
		bExecute := TRUE,
		sJsonPathName := 'C:\PLCUtility\CalDat_Powerstack.json',
		sStructName := 'ST_System_Calibration',
		pStruct := ADR(settings.Calibration),
		nStruct := SIZEOF(settings.Calibration),
		WriteMode := FALSE,
		sMessage => sMessage
		);
	ELSE
		SFCstep := 0;
		rTrigExecute(CLK := FALSE);
		StoreSettings := TRUE;	
END_CASE


IF b_next THEN 
	tDelaySFCstep(IN := TRUE);
 	IF tDelaySFCstep.q THEN 
	SFCstep := SFCstep + 1;
		tDelaySFCstep(IN := FALSE);
	END_IF 
END_IF
END_METHOD

METHOD UpdateSystemTime : BOOL
VAR_INST
	SetTime :	NT_SetLocalTime();
	rtrig_AutoUpdate	:	r_Trig;
	ftrig_UpdateDone	:	f_Trig;
	systime				:	Timestruct;

	SystemTimeStamp		:	DINT;
	GPSTimeStamp		:	DINT;
	TON_GpsUpdateReq	:	TON := (PT := T#5M); 
	
	NewTimeString		:	STRING;
	NewTimeStruct		:	Timestruct;

	
	UpdateRequired		:	BOOL;
END_VAR

monitor.system.DT_SystemTime := GVL.dt_SystemDateTime;

//first fix datetime format from teltonika.
IF st_params.SystemTime.AutoSyncToGPS THEN 
	TON_GpsUpdateReq(in := ABS(DT_TO_DINT(monitor.router.GPS.DateTime) - DT_TO_DINT(gvl.dt_SystemDateTime)) > 30);
	IF ton_gpsUpdateReq.Q THEN
		NewTimeStruct := DT_TO_Systemtime(monitor.Router.GPS.DateTime);
		UpdateRequired	:=	TRUE;
	ELSE
		UpdateRequired	:=	FALSE;
	END_IF
ELSE
	IF st_params.SystemTime.ManualSync THEN
		st_params.SystemTime.ManualSync := FALSE;
		NewTimeStruct := DT_TO_SYSTEMTIME(st_params.SystemTime.ManSyncValue);
		UpdateRequired	:=	TRUE;
	END_IF
END_IF
	
SetTime(	TimeSTR := NewTimeStruct, //convert to Systemtime struct and write to plc
	start	:= UpdateRequired,
	TMOUT	:= T#1S);

			
ftrig_UpdateDone(clk := SetTime.BUSY);

IF ftrig_UpdateDone.Q THEN
	UpdateRequired := FALSE;
	monitor.system.events.b_TimeUpdateFailed := FALSE;
	IF SetTime.ERR THEN
		monitor.system.events.b_TimeUpdateFailed := TRUE;
	END_IF
END_IF
END_METHOD

END_FUNCTION_BLOCK

(* stored: Version 1.1.0.1, ProductVersion 3.1.4026.18
   POU FB_SystemControl: Id {80088fce-282f-4b1a-b9ec-9bb5f8a72aa2}, SpecialFunc None
   Folder MapUserControls: Id {e317cc20-b8c7-40c1-90fb-f89a885a87cd}
   Folder Nested Methods: Id {91f678d8-34d0-4f15-851f-53116a7d863f}
   Folder CalibrationData: Id {4a10be61-d1c6-4857-bb52-89910a20f797}
   Method CalculateEfficiency: Id {b9132480-21ec-4ac3-8cdc-f0a527c48fe2}
   Method ConfigureOutputContact: Id {4e9210a3-d285-4c3d-bd99-cd0cd99c0a84}
   Method EMstop: Id {604c76fd-14d0-4f9f-9eed-a29665787efd}
   Method FillSystemMonitoringVars: Id {960a52bb-9693-4a14-9722-711dbd0dc6dd}
   Method GetDiagnostics: Id {d9c5c631-8daf-4557-b7ee-b75fbce17ea6}
   Method GetEvents: Id {3333007a-2c08-44e7-9058-6a89010670fd}
   Method JsonFileToStruct: Id {3da0cc58-6182-449d-ad88-97a711d43219}
   Action Map_ACDCchargerControls: Id {157f25bb-449d-4952-b509-1819c294357b}
   Action MaP_BMSControl: Id {22b5f460-c89a-4b43-bc7d-f91c8855495d}
   Action Map_DCLink: Id {c790f86f-095a-4d2d-9245-c022de359acc}
   Action Map_GenCommControls: Id {caba063b-ae87-4540-8f08-a9ef67027d59}
   Action Map_GeneralControls: Id {f60fee37-1a84-40c2-9e3c-a2a9a227edc1}
   Action Map_HartingIO: Id {3458e5ed-6acb-42c3-9faf-2b81378bffd7}
   Action Map_PowerstackControls: Id {f49c1718-94cd-4aa2-9d51-e0b9de4e098e}
   Action Map_ProtectionSystemControls: Id {ee73439e-2460-4b96-9ca4-c82871edbc64}
   Action Map_PSBControls: Id {a0999be7-db6d-4861-93ec-ed2833fab5c7}
   Method MapUsercontrolsToSystemVars: Id {b06c8f50-2f97-4eb7-80bb-658f05e084d1}
   Method PowerstackCalibration: Id {8b81fc85-34cc-4f1d-81f1-6ff0da9baa8c}
   Method Reset: Id {ad65bbc2-7efb-47ba-b576-ea2f90bb992f}
   Method SetPQLimits: Id {0a2e50ba-aca0-428c-a77c-a40ef6705f6c}
   Method shutdown: Id {d476ef20-e6dd-456d-9d5b-e628a2578fb8}
   Method StoreSettings: Id {213388af-3df9-4880-9930-c0e2dce77aca}
   Method UpdateSystemTime: Id {c3cb0c87-8a74-4cfc-a557-923712f0b417} *)
